DATA_BLOCK "InstAnalyzeTokens2"
{ S7_Optimized_Access := 'TRUE' }
AUTHOR : 'SIEMENS AG'
VERSION : 3.0
NON_RETAIN
"AnalyzeTokens"

BEGIN

END_DATA_BLOCK

